RoboDK station: nithin hack1.rdk

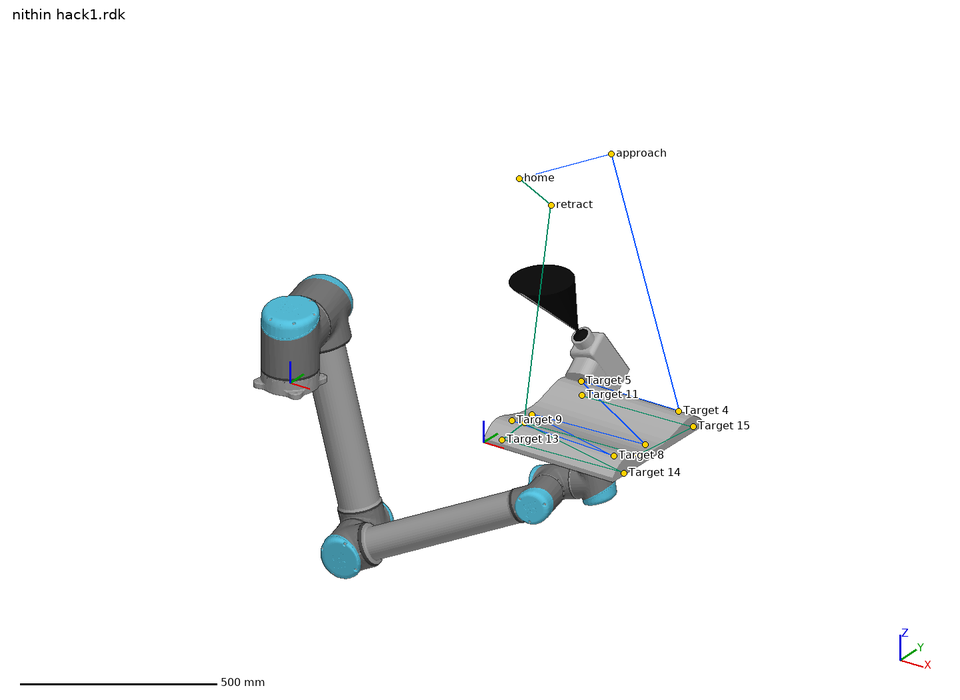
[picture v0: the station drawn from its stored meshes, robots at their saved joint values, targets as dots, program paths as lines]
Station nithin hack1 (saved by RoboDK 5.7.3). Poses are relative to the parent item; angles as X-Y-Z fixed-axis rotations.
  - frame UR10 Base at (0, 0, 0) mm
    - robot UR10: 6 axes, payload 10 kg, reach 1300 mm, repeatability 0.1 mm, weight 28.9 kg
        modified DH rows (alpha deg, a mm, theta deg, d mm): 0, 0, 0, 128; 90, 0, 180, 0; 0, 612.7, 0, 0; 0, 571.6, 0, 163.9; -90, 0, 0, 115.7; 90, 0, 180, 92.2
        joint limits [-360, -360, -360, -360, -360, -360] to [360, 360, 360, 360, 360, 360]; home [0, -90, -90, 0, 90, 0]; saved at [193.684, 77.103, -101.168, -78.418, 86.987, 166.645]
      - tool Paint gun, TCP at (0, 0, 200) mm, size 277.6 x 203.2 x 501.7 mm, geometry from Paint gun.stl
  - frame Frame 2 at (600, 0, 0) mm
    - object Object Inspection at (0, 0, 0) mm, size 400 x 400 x 46.2 mm, geometry from Object Inspection.stl
    - target home (Cartesian target) at (20, 129.35, 700.58) mm, rotated rx 121.94 ry 0 rz -90 deg; joints [177.712, -15.576, -38.774, -157.609, 91.941, 178.789] of UR10
    - target approach (Cartesian target) at (71.66, 462.7, 651.41) mm, rotated rx -177.34 ry 21.09 rz -76.59 deg; joints [44.279, -99.354, -82.879, -74.242, 106.548, 33.334] of UR10
    - target retract (Cartesian target) at (155.17, 78.27, 683.41) mm, rotated rx -177.25 ry 25.7 rz -76.35 deg; joints [15.326, -95.315, -82.625, -88.209, 115.569, 3.175] of UR10
    - target Target 4 (Cartesian target) at (350.35, 364.41, 40.88) mm, rotated rx 170.94 ry -24.03 rz -68.62 deg; joints [32.174, -140.133, -79.959, -64.214, 68.556, 15.451] of UR10
    - target Target 5 (Cartesian target) at (43.8, 369.83, 38.29) mm, rotated rx 170.94 ry -24.03 rz -68.62 deg; joints [44.871, -122.829, -115.101, -50.739, 72.176, 28.379] of UR10
    - target Target 8 (Cartesian target) at (370.35, 50.02, 45.05) mm, rotated rx -173.21 ry 9.32 rz -53.69 deg; joints [11.585, -137.024, -89.533, -41.101, 101.277, -23.94] of UR10
    - target Target 9 (Cartesian target) at (40.72, 66.69, 45.77) mm, rotated rx 178.83 ry -1.58 rz -53.46 deg; joints [20.954, -118.231, -129.37, -23.102, 88.163, -15.553] of UR10
    - target Target 8 (Cartesian target) at (366.07, 194.53, 18.37) mm, rotated rx 179.88 ry -0.48 rz -76.29 deg; joints [21.002, -139.322, -87.444, -43.411, 89.539, 7.294] of UR10
    - target Target 9 (Cartesian target) at (31.83, 169.55, 19.94) mm, rotated rx 178.02 ry -7.98 rz -76.03 deg; joints [30.56, -121.038, -127.872, -25.291, 82.927, 16.99] of UR10
    - target Target 11 (Cartesian target) at (49.11, 366.79, 0) mm, rotated rx 0 ry 0 rz -90 deg; joints [42.168, -153.807, -85.326, 149.133, 90, -42.168] of UR10
    - target Target 12 (Cartesian target) at (362.32, 167.46, 0) mm, rotated rx 0 ry 0 rz -90 deg; joints [19.531, -170.68, -43.294, 123.975, 90, -19.531] of UR10
    - target Target 13 (Cartesian target) at (29.4, 39.86, 0) mm, rotated rx 0 ry 0 rz -90 deg; joints [18.687, -149.01, -100.568, 159.578, 90, -18.687] of UR10
    - target Target 14 (Cartesian target) at (393.94, 60.03, 0) mm, rotated rx 0 ry 0 rz -90 deg; joints [12.93, -173.009, -38.035, 121.044, 90, -12.93] of UR10
    - target Target 14 (Cartesian target) at (49.11, 366.79, 0) mm, rotated rx 0 ry 0 rz -90 deg; joints [42.168, -153.807, -85.326, 149.133, 90, -42.168] of UR10
    - target Target 15 (Cartesian target) at (384.45, 380.79, 0) mm, rotated rx 0 ry 0 rz -90 deg; joints [30.08, -185.609, -10.679, 106.288, 90, -30.08] of UR10
    - target Target 16 (Cartesian target) at (20.15, 152.94, 0) mm, rotated rx 0 ry 0 rz -90 deg; joints [28.722, -149.291, -99.556, 158.848, 90, -28.722] of UR10
  - program Prog1 (9 instructions, listed below)
  - program retract move (3 instructions, listed below)
  - program MainProgram (11 instructions, listed below)
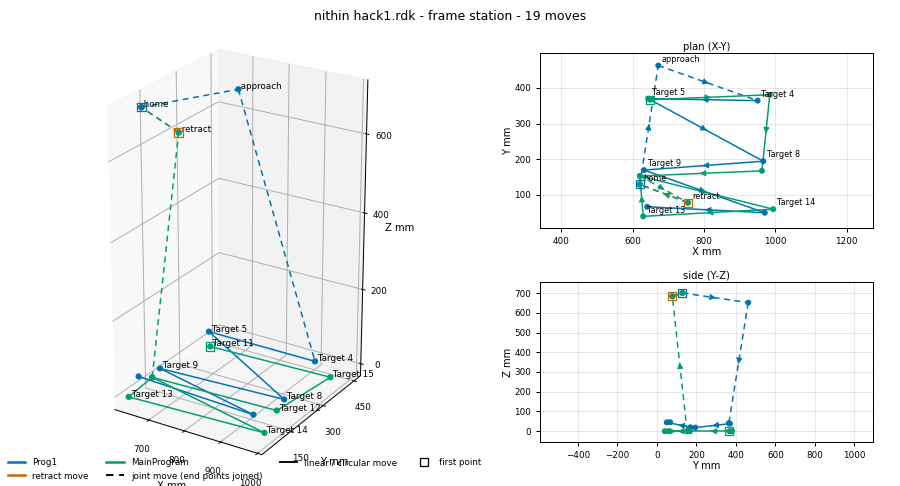
[picture p0: tool path of nithin hack1.rdk in frame station, 19 of 19 moves have a stored position in this frame; points joined in program order, loops and branches not executed]

--- program Prog1 (robot UR10) ---
  Set Ref.: Frame 2
  MoveJ (home)
  MoveJ (approach)
  MoveJ (Target 4)
  MoveL (Target 5)
  MoveL (Target 8)
  MoveL (Target 9)
  MoveL (Target 8)
  MoveL (Target 9)

--- program retract move (robot UR10) ---
  Set Ref.: Frame 2
  MoveJ (retract)
  MoveJ (home)

--- program MainProgram (robot UR10) ---
  Call Prog1
  Call retract move
  MoveL (Target 11)
  MoveL (Target 15)
  MoveL (Target 12)
  MoveL (Target 16)
  MoveL (Target 14)
  MoveL (Target 13)
  MoveL (Target 16)
  MoveJ (retract)
  MoveJ (home)
